{attribute 'qualified_only'}
VAR_GLOBAL
	isResetON	: BOOL;
	isStopON	: BOOL;
	isEmgStopON	: BOOL;
	
END_VAR

(* stored: Version 1.1.0.1, ProductVersion 3.1.4024.12
   GVL GVL_System: Id {9d484d26-0ed9-4a22-840b-fd35cf8e32ed} *)
